// TIA Portal V20 export
VAR_GLOBAL   // PLC tag table "Default tag table"
   Sick_Sensor_Vlaue AT %IW64 : Int;
   RealValue AT %MD10 : Real;
   finalValue AT %MD14 : Real;
   Tag_1 AT %MD20 : Real;
   Out_1 AT %Q0.0 : Bool;
   Activ AT %I0.0 : Bool;
   Out_2 AT %Q0.1 : Bool;
   Tag_5 AT %M0.0 : Bool;
   Out_4 AT %Q0.3 : Bool;
   System_Byte AT %MB1 : Byte;
   FirstScan AT %M1.0 : Bool;
   DiagStatusUpdate AT %M1.1 : Bool;
   AlwaysTRUE AT %M1.2 : Bool;
   AlwaysFALSE AT %M1.3 : Bool;
   Tag_7 AT %M100.0 : Bool;
   Sen_3 AT %IW10 : Int;
   Sen_4 AT %IW12 : Int;
   Sen_5 AT %IW14 : Int;
   Sen_6 AT %IW16 : Int;
   Tag_8 AT %M20.0 : Bool;
   Tag_9 AT %M30.5 : Bool;
   Clock_Byte AT %MB100 : Byte;
   Clock_10Hz AT %M100.0 : Bool;
   Clock_5Hz AT %M100.1 : Bool;
   "Clock_2.5Hz" AT %M100.2 : Bool;
   Clock_2Hz AT %M100.3 : Bool;
   "Clock_1.25Hz" AT %M100.4 : Bool;
   Clock_1Hz AT %M100.5 : Bool;
   "Clock_0.625Hz" AT %M100.6 : Bool;
   "Clock_0.5Hz" AT %M100.7 : Bool;
   Tag_10 AT %M7.7 : Bool;
   Tag_11 AT %M7.1 : Bool;
   Tag_12 AT %M2.2 : Bool;
   inter_segnal AT %M2.0 : Bool;
   Error_i AT %I0.1 : Bool;
   Reset_Error AT %I0.2 : Bool;
   Tag_2 AT %MW20 : Int;
   Tag_3 AT %MD30 : Real;
   Tag_4 AT %MD31 : Real;
   Out_3 AT %Q0.2 : Bool;
   Out_5 AT %Q0.4 : Bool;
   Out_6 AT %Q0.5 : Bool;
   Out_7 AT %Q0.6 : Bool;
   Out_8 AT %Q0.7 : Bool;
   Out_9 AT %Q1.0 : Bool;
   Out_10 AT %Q1.1 : Bool;
   Tag_6 AT %M40.1 : Bool;
   Tag_13 AT %MD33 : DWord;
   Tag_14 AT %M32.1 : Bool;
   Tag_15 AT %M32.2 : Bool;
   "Wire-break-Error" AT %M90.1 : Bool;
   SEN_Freigabe AT %M90.2 : Bool;
   "System_Byte(1)" AT %MB10 : Byte;
   Tag_16 AT %M0.5 : Bool;
   Tag_17 AT %M11.1 : Bool;
END_VAR
